FUNCTION_BLOCK PUBLIC FB_Machine IMPLEMENTS I_StateMachine
VAR_INPUT
	bButton				: BOOL;
	bInsertCoin			: BOOL;
	bTakeProduct 		:	BOOL;
	bTakeCoin 			:	BOOL;	
END_VAR
VAR_OUTPUT
	ipState				:	I_State := fbWaitingState;	
		
END_VAR
VAR
	fbCoinEjectedState		:	FB_CoinEjectedState;
	fbHasCoinState				:	FB_HasCoinState;
	fbProductEjectedState	:	FB_ProductEjectedState;
	fbWaitingState				:	FB_WaitingState;
	
	_nProducts			:	UINT;
	
	rtrigButton				:	R_TRIG;
	rtrigInsertCoin			:	R_TRIG;
	rtrigTakeProduct		:	R_TRIG;
	rtrigTakeCoin			:	R_TRIG;
END_VAR

rtrigButton(CLK := bButton);
rtrigInsertCoin(CLK := bInsertCoin);
rtrigTakeProduct(CLK := bTakeProduct);
rtrigTakeCoin(CLK := bTakeCoin);

IF (rtrigButton.Q) THEN
	ipState.PressButton();
END_IF

IF (rtrigInsertCoin.Q) THEN
	ipState.InsertCoin();
END_IF

IF (rtrigTakeProduct.Q) THEN
	ipState.CustomerTakesProduct();
END_IF

IF (rtrigTakeCoin.Q) THEN
	ipState.CustomerTakesCoin();
END_IF

PROPERTY INTERNAL CoinEjectedState : I_State
GET
CoinEjectedState := THIS^.fbCoinEjectedState;
END_GET
END_PROPERTY

METHOD FB_init : BOOL
VAR_INPUT
	bInitRetains : BOOL; // if TRUE, the retain variables are initialized (warm start / cold start)
	bInCopyCode : BOOL;  // if TRUE, the instance afterwards gets moved into the copy code (online change)
	nProducts :	UINT;
END_VAR
THIS^._nProducts := nProducts;

wireUpStateTransitions();
END_METHOD

PROPERTY INTERNAL HasCoinState : I_State
GET
HasCoinState := THIS^.fbHasCoinState;
END_GET
END_PROPERTY

PROPERTY INTERNAL nProducts : UINT
GET
nProducts := _nProducts;
END_GET
END_PROPERTY

PROPERTY INTERNAL ProductEjectedState : I_State
GET
ProductEjectedState := THIS^.fbProductEjectedState;
END_GET
END_PROPERTY

METHOD INTERNAL SetProducts : BOOL
VAR_INPUT
	newProducts : UINT;
END_VAR
THIS^._nProducts := newProducts;
END_METHOD

METHOD INTERNAL SetState : BOOL
VAR_INPUT
	newState : I_State;
END_VAR
THIS^.ipState := newState;
END_METHOD

PROPERTY INTERNAL WaitingState : I_State
GET
WaitingState := THIS^.fbWaitingState;
END_GET
END_PROPERTY

METHOD PRIVATE wireUpStateTransitions
fbWaitingState.SetTransitionStates(
	Machine := THIS^,
	CoinInsertedNext := fbHasCoinState
);

fbHasCoinState.SetTransitionStates(
	Machine := THIS^,
	ButtonPressedProductDecrementedNext := fbProductEjectedState,
	ButtonPressedNoProductNext := fbCoinEjectedState
);

fbProductEjectedState.SetTransitionStates(
	Machine := THIS^,
	AfterProductEjectedNext := fbWaitingState
);

fbCoinEjectedState.SetTransitionStates(
	Machine := THIS^,
	CustomerTakesCoinNext := fbWaitingState
);
END_METHOD

END_FUNCTION_BLOCK

(* stored: Version 1.1.0.1, ProductVersion 3.1.4022.17
   POU FB_Machine: Id {f50e73cc-6d6c-4918-b2bc-262d6ffb1bde}, SpecialFunc None
   Property CoinEjectedState: Id {3bae123f-1761-4dcd-8840-7f4f4dc8ca19}
   Get Get: Id {5e73377e-92d7-4e7c-bc4b-1dd9540c5295}
   Method FB_init: Id {a213588c-99e9-403d-b664-265c20a195d3}
   Property HasCoinState: Id {1c464c53-5fcc-473d-971b-69693b0a5e63}
   Get Get: Id {245a105b-8b85-4d11-a9f1-08b0b7979c28}
   Property nProducts: Id {975c93c0-dd8a-466a-8e50-ab97cdd99152}
   Get Get: Id {41353718-922a-43d3-9b0d-14698c0e66ad}
   Property ProductEjectedState: Id {3d47f721-b04c-4fca-90ae-11edfaf5352d}
   Get Get: Id {5a5f582c-330b-4650-974a-35fdfda8f2b6}
   Method SetProducts: Id {aabe1e3c-336b-476b-b3f0-3aa38b51e028}
   Method SetState: Id {bac7998a-96e0-484d-9b0b-984b4f2ae380}
   Property WaitingState: Id {50c40cfc-35ec-45fa-bb16-115c583a60c7}
   Get Get: Id {b4d9b6ac-64a3-4669-8d92-757ed4ecacb1}
   Method wireUpStateTransitions: Id {ae777051-a0ea-4107-b4e5-d78929e86b79} *)
